// Mitsubishi GX Works2 project: BKVinaTest   PLC: FX3U/FX3UC

// global labels: Global1
VAR_GLOBAL
  ALARM AT Y012 : BOOL;
  OPERATION AT Y013 : BOOL;
  RelayXLKC1 AT Y014 : BOOL;
  RelayXLC2 AT Y015 : BOOL;
  RelayXLD3_1 AT Y016 : BOOL;
  RelayXLD3_2 AT Y017 : BOOL;
  RelayXLX4_1 AT Y020 : BOOL;
  RelayXLX4_2 AT Y021 : BOOL;
  RelayXLX5_1 AT Y022 : BOOL;
  RelayXLX5_2 AT Y023 : BOOL;
  RelayXLD6_1 AT Y024 : BOOL;
  RelayLubOil AT Y025 : BOOL;
  RelayXLTT AT Y026 : BOOL;
  RelayXLTP AT Y027 : BOOL;
  RelayXLDT AT Y030 : BOOL;
  RelayXLDP AT Y031 : BOOL;
  RelayXLKDT AT Y032 : BOOL;
  RelayXLKDP AT Y033 : BOOL;
  RelayTT AT Y034 : BOOL;
  RelayMR_1 AT Y035 : BOOL;
  RelayMR_2 AT Y036 : BOOL;
  RelayMXC_1 AT Y037 : BOOL;
  RelayMXC_2 AT Y040 : BOOL;
  RelayMQ_1 AT M10 : BOOL;
  RelayMQ_2 : BOOL;
  RelayMXDT_1 AT Y041 : BOOL;
  RelayMXDT_2 AT Y042 : BOOL;
  RelayMXDP_1 AT Y043 : BOOL;
  RelayMXDP_2 AT Y044 : BOOL;
  RelayOilP AT Y045 : BOOL;
  RelayOilV1 AT Y046 : BOOL;
  RelayOilV2 AT Y047 : BOOL;
  CommandMXC_F AT M260 : BOOL;
  CommandMXC_Z AT M261 : BOOL;
  CommandMQ_F AT M262 : BOOL;
  CommandMQ_Z AT M263 : BOOL;
  CommandMXDT_F AT M264 : BOOL;
  CommandMXDT_Z AT M265 : BOOL;
  CommandMXDP_F AT M267 : BOOL;
  CommandMXDP_Z AT M268 : BOOL;
  CommandMR_L AT M269 : BOOL;
  CommandMR_R AT M270 : BOOL;
  CommandXLXC_I AT M271 : BOOL;
  CommandXLXC_O AT M272 : BOOL;
  CommandPHA_1 AT M273 : BOOL;
  CommandPHA_2 AT M274 : BOOL;
  MR_L AT X010 : BOOL;
  MR_R AT X011 : BOOL;
  CB3 AT X012 : BOOL;
  EMERG AT X013 : BOOL;
  MainRST AT X014 : BOOL;
  START AT X015 : BOOL;
  Jog_Left AT X016 : BOOL;
  Jog_Right AT X017 : BOOL;
  PushOilPump AT X020 : BOOL;
  XLKC1_I AT X021 : BOOL;
  XLKC1_O AT X022 : BOOL;
  XLC2_I AT X023 : BOOL;
  XLC2_O AT X024 : BOOL;
  XLD3_I AT X025 : BOOL;
  XLD3_O AT X026 : BOOL;
  XLX4_I AT X027 : BOOL;
  XLX4_O AT X030 : BOOL;
  XLX5_I AT X031 : BOOL;
  XLX5_O AT X032 : BOOL;
  XLD6_I AT X033 : BOOL;
  XLD6_O AT X034 : BOOL;
  XLTT_I AT X035 : BOOL;
  XLTP_I AT X036 : BOOL;
  XLKDT_I AT X037 : BOOL;
  XLKDP_I AT X040 : BOOL;
  XLDT_I AT X041 : BOOL;
  XLDT_O AT X042 : BOOL;
  XLDP_I AT X043 : BOOL;
  XLDP_O AT X044 : BOOL;
  OLPump AT X045 : BOOL;
  MR_L1 AT X046 : BOOL;
  MR_R1 AT X047 : BOOL;
  MXC_ZX AT X004 : BOOL;
  MQ_ZX AT X005 : BOOL;
  MXDT_ZX AT X002 : BOOL;
  MXDP_ZX AT X003 : BOOL;
  Round_MXC AT D200 : REAL;
  Round_MQL AT D202 : REAL;
  Round_MQR AT D204 : REAL;
  Round_MXDT AT D206 : REAL;
  Round_MXDP AT D208 : REAL;
  CommandBTX AT M275 : BOOL;
  CommandXLTT AT M276 : BOOL;
  CommandXLTP AT M277 : BOOL;
  CommandXLDT AT M278 : BOOL;
  CommandXLDP AT M279 : BOOL;
  CommandXLKC1 AT M280 : BOOL;
  CommandXLC2 AT M281 : BOOL;
  MXC_Z AT M282 : BOOL;
  MQ_Z AT M283 : BOOL;
  MXDT_Z AT M284 : BOOL;
  MXDP_Z AT M285 : BOOL;
  MXC_FWD AT M286 : BOOL;
  MQ_FWD AT M287 : BOOL;
  MXDT_FWD AT M288 : BOOL;
  MXDP_FWD AT M289 : BOOL;
  ModeAuto : BOOL;
  StopEmerg : BOOL;
  activeCK : BOOL;
  pushManXLKC1 AT M200 : BOOL;
  pushManXLC2 AT M201 : BOOL;
  pushManXLD3_I AT M202 : BOOL;
  pushManXLD3_O AT M203 : BOOL;
  pushManXLX4_I AT M204 : BOOL;
  pushManXLX4_O AT M205 : BOOL;
  pushManXLX5_I AT M206 : BOOL;
  pushManXLX5_O AT M207 : BOOL;
  pushManXLD6_I AT M208 : BOOL;
  pushManXLD6_O AT M209 : BOOL;
  pushManXLTT AT M210 : BOOL;
  pushManXLTP AT M211 : BOOL;
  pushManXLKDT AT M212 : BOOL;
  pushManXLKDP AT M213 : BOOL;
  pushManXLDT AT M214 : BOOL;
  pushManXLDP AT M215 : BOOL;
  pushManTT AT M216 : BOOL;
  pushManMXC_F AT M217 : BOOL;
  pushManMXC_Z AT M218 : BOOL;
  pushManMQ_F AT M219 : BOOL;
  pushManMQ_Z AT M220 : BOOL;
  pushManMXDT_F AT M221 : BOOL;
  pushManMXDT_Z AT M222 : BOOL;
  pushManMXDP_F AT M223 : BOOL;
  pushManMXDP_Z AT M224 : BOOL;
  PushOilV1 AT M225 : BOOL;
  PushOilV2 AT M226 : BOOL;
  pushB8 AT M227 : BOOL;
  pushB9 AT M228 : BOOL;
  pushB10 AT M229 : BOOL;
  pushCa1 AT M230 : BOOL;
  pushCa2 AT M231 : BOOL;
  pushCa3 AT M232 : BOOL;
  rstTotalB AT M233 : BOOL;
  rstCounterCK AT M234 : BOOL;
  rstAmountCK AT M235 : BOOL;
  restory AT M236 : BOOL;
  Round_MR AT D210 : REAL;
  Speed_MXC AT D212 : REAL;
  Speed_MQ AT D214 : REAL;
  Speed_MXDT AT D216 : REAL;
  Speed_MXDP AT D218 : REAL;
  Speed_MR AT D220 : REAL;
  Speed_MXCZ AT D222 : REAL;
  Speed_MQZ AT D224 : REAL;
  Speed_MXDTZ AT D226 : REAL;
  Speed_MXDPZ AT D228 : REAL;
  Speed_MRZ AT D230 : REAL;
  Real_MXC : REAL;
  Real_MQ : REAL;
  Real_MXDT : REAL;
  Real_MXDP : REAL;
  Real_MR : REAL;
  Freq_MXC : REAL;
  Freq_MQ : REAL;
  Freq_MXDT : REAL;
  Freq_MXDP : REAL;
  Freq_MR : REAL;
  TimeMR_DSL AT D240 : DWORD;
  TimeMR_R AT D242 : DWORD;
  TimeMR_E AT D244 : DWORD;
  TimeERROR AT D246 : DWORD;
  MXCF1 AT Y000 : BOOL;
  MXCE1 AT Y001 : BOOL;
  MXCD1 AT Y002 : BOOL;
  MR_DSLOW AT Y011 : BOOL;
  ca1_B8 AT D250 : DWORD;
  ca2_B8 AT D252 : DWORD;
  ca3_B8 AT D254 : DWORD;
  ca1_B9 AT D256 : DWORD;
  ca2_B9 AT D258 : DWORD;
  ca3_B9 AT D260 : DWORD;
  ca1_B10 AT D262 : DWORD;
  ca2_B10 AT D264 : DWORD;
  ca3_B10 AT D266 : DWORD;
  total_B8 AT D268 : DWORD;
  total_B9 AT D270 : DWORD;
  total_B10 AT D272 : DWORD;
  NumberCK AT D280 : DWORD;
  CounterCK AT D282 : DWORD;
  AmountCK AT D284 : DWORD;
  TotalCK AT D286 : DWORD;
  PushLubOil AT M237 : BOOL;
  Pape1 AT M240 : BOOL;
  Pape2 AT M241 : BOOL;
  Pape3 AT M242 : BOOL;
  PushPause AT M238 : BOOL;
  Pape0 AT M239 : BOOL;
  IndicateMXC AT D232 : REAL;
  IndicateMQ AT D234 : REAL;
  IndicateMXDT AT D236 : REAL;
  IndicateMXDP AT D238 : REAL;
END_VAR

// task Task_01 (event TRUE, interval 0, priority 31): PowerControl, StepControl
// task InterruptMXC (event I010, interval 0, priority 31): EncoderX001
// task InterruptMXDT (event I020, interval 0, priority 31): EncoderX006
// task InterruptMXDP (event I030, interval 0, priority 31): EncoderX007
// task InterruptMQ_Z (event I501, interval 0, priority 31): PickupX005
// task InterruptMXC_Z (event I400, interval 0, priority 31): PickupX004
// task InterruptMXDT_Z (event I200, interval 0, priority 31): PickupX002
// task InterruptMXDP_Z (event I300, interval 0, priority 31): PickupX003

PROGRAM PowerControl
VAR
  ButtonOilP : BOOL;
  ButtonOilV1 : BOOL;
  ButtonOilV2 : BOOL;
  MR : MotorRev;
  MQ : MotorRev;
  MXC : MotorRev;
  MXDT : MotorRev;
  MXDP : MotorRev;
  XLKC1 : MotorOne;
  XLC2 : MotorOne;
  XLD3 : MotorRev;
  XLX4 : MotorRev;
  XLX5 : MotorRev;
  XLD6 : MotorOne;
  XLTT : MotorOne;
  XLTP : MotorOne;
  XLKDT : MotorOne;
  XLKDP : MotorOne;
  XLDT : MotorOne;
  XLDP : MotorOne;
  OILPUMP : MotorOne;
  VALVE1 : MotorOne;
  VALVE2 : MotorOne;
  Servo_MXC : Servo;
  TimerMR_DSL : TON;
  TimerMRDSL_Q : BOOL;
  ManualMXC_F : BOOL;
  ManualMXC_Z : BOOL;
  ManualMQ_F : BOOL;
  ManualMQ_Z : BOOL;
  ManualMXDT_F : BOOL;
  ManualMXDT_Z : BOOL;
  ManualMXDP_F : BOOL;
  ManualMXDP_Z : BOOL;
  Dint_C251 : DINT;
  Dint_C234 : DINT;
  Dint_C244 : DINT;
  Dint_C245 : DINT;
END_VAR
EI( TRUE );
(* MR: Chạy khi cụm xoắn đầu chạy *)
MR(SetAutoMan := ModeAuto, PushManF := Jog_Left , PushManR := Jog_Right ,
		LimitInputF := NOT MR_L OR NOT TimerMRDSL_Q, LimitInputR := NOT MR_R OR NOT TimerMRDSL_Q,
		SetAutoRunF := CommandMR_L, SetAutoRunR := CommandMR_R ,
		OutputF := RelayMR_1, OutputR:= RelayMR_2);

RelayTT := (RelayMR_1 AND NOT MR_L) OR (RelayMR_2 AND NOT MR_R);
TimerMR_DSL(IN := (NOT MR_L AND RelayMR_1) OR (NOT MR_R AND RelayMR_2), 
								PT := DWORD_TO_TIME(TimeMR_DSL), Q := TimerMRDSL_Q );

SET(LDP(TRUE, (MR_L1 AND RelayMR_1) OR (MR_R1 AND RelayMR_2)), MR_DSLOW);
RST(LDP(TRUE, RelayMR_1 OR RelayMR_2), MR_DSLOW);

(* MXQ: *)
(* Initialize FX2N-1HC => MQ control *)
TO( M8002, K0, K0 , K0, K1 );
DTO( M8002, K2147483647, K0 , K2, K1 );
DTO( M8002 , REAL_TO_DINT( Real_MQ ) , K0, K12 , K1);

M11 := ModeAuto;
M13 := ModeAuto;
M10 := CommandMQ_F OR pushManMQ_F;
M14 := NOT M10;
SET( LDP(TRUE, M10), M22); (*YS output set *)
RST( LDF(TRUE, M34), M8055);
RST( LDF(TRUE, M34), CommandMQ_F);

TO( TRUE, K4M10, K0 , K4, K1 );
DFROM( TRUE, K0 , K20 , K1, C234 );
FROM( ModeAuto, K0 , K27 , K1 , K3M30 );
DTO( LDF(TRUE, M10) , K0 , K0, K20 , K1); (* software reset counter *)

(*Manual*)	

RST( LDF(TRUE , NOT ModeAuto AND pushManMQ_F), M20); (*YS output reset*)
	
(* MXC:  CommandXLXC_I  and CommandXLXC_O *)	
SET( LDP(TRUE, XLD3_O AND XLX4_O), CommandMXC_F);
MXC(SetAutoMan:= ModeAuto, PushManF := pushManMXC_F, 
			LimitInputF := MXC_FWD, LimitInputR := MXC_Z,
			SetAutoRunF := CommandMXC_F, SetAutoRunR := CommandMXC_Z,
			OutputF := RelayMXC_1, OutputR := RelayMXC_2);

RST( LDP(TRUE, CommandXLXC_O), CommandXLXC_I);
RST( LDF(TRUE, CommandMXC_Z), CommandXLXC_O);
SET( LDF(TRUE, CommandMXC_Z), CommandXLXC_I);
XLD3(SetAutoMan := ModeAuto,
			PushManF := pushManXLD3_O, PushManR := pushManXLD3_I,
			LimitInputF := TRUE, LimitInputR := TRUE,
			SetAutoRunF := CommandXLXC_O, SetAutoRunR := CommandXLXC_I,
			OutputF := RelayXLD3_1, OutputR := RelayXLD3_2);			
			
XLX4(SetAutoMan := ModeAuto,
			PushManF := pushManXLX4_O, PushManR := pushManXLX4_I,
			LimitInputF := TRUE , LimitInputR := TRUE,
			SetAutoRunF := CommandXLXC_O, SetAutoRunR := CommandXLXC_I,
			OutputF := RelayXLX4_1, OutputR := RelayXLX4_2);				
	
(* MXDT:  CommandXLDT => dừng khi encoder đủ vòng *)	
SET( LDP(TRUE, XLDT_O), CommandMXDT_F);
SET( LDP(TRUE, XLDT_I), CommandMXDT_Z);
MXDT(SetAutoMan := ModeAuto, PushManF := pushManMXDT_F, 
			LimitInputF := MXDT_FWD, LimitInputR := MXDT_Z,
			SetAutoRunF :=  CommandMXDT_F, SetAutoRunR := CommandMXDT_Z ,
			OutputF := RelayMXDT_1, OutputR := RelayMXDT_2);

RST( LDF(TRUE, MXDT_FWD), CommandXLDT);
XLKDT(SetAutoMan := ModeAuto, 
			PushMan := pushManXLKDT, LimitInput :=  TRUE,
			SetAutoRun := CommandXLDT, Output := RelayXLKDT);

XLDT(SetAutoMan := ModeAuto, 
			PushMan := pushManXLDT, LimitInput :=TRUE,
			SetAutoRun := CommandXLDT, Output := RelayXLDT);	

(* MXDP:  CommandXLDP => dừng khi encoder đủ vòng *)	
SET( LDP(TRUE, XLDP_O), CommandMXDP_F);
SET( LDP(TRUE, XLDP_I), CommandMXDP_Z);
MXDP(SetAutoMan := ModeAuto, PushManF := pushManMXDP_F, 
			LimitInputF := MXDP_FWD, LimitInputR := MXDP_Z,
			SetAutoRunF := CommandMXDP_F, SetAutoRunR := CommandMXDP_Z ,
			OutputF := RelayMXDP_1, OutputR := RelayMXDP_2);

RST( LDF(TRUE, MXDP_FWD), CommandXLDP);
XLKDP(SetAutoMan := ModeAuto, 
			PushMan := pushManXLKDP, LimitInput := TRUE,
			SetAutoRun := CommandXLDP, Output := RelayXLKDP);
			
XLDP(SetAutoMan := ModeAuto,
			PushMan := pushManXLDP, LimitInput := TRUE,
			SetAutoRun := CommandXLDP, Output := RelayXLDP);

(* PHA:  CommandPHA_1  and CommandPHA_2 *)	
SET(LDP(TRUE, MR_R AND CommandBTX), CommandPHA_1);
SET(LDP(TRUE, MR_L AND CommandBTX), CommandPHA_2);	
XLX5(SetAutoMan := ModeAuto,
			PushManF := pushManXLX5_O, PushManR := pushManXLX5_I,
			LimitInputF := TRUE , LimitInputR := TRUE,
			SetAutoRunF := CommandPHA_1, SetAutoRunR := CommandPHA_2,
			OutputF := RelayXLX5_1, OutputR := RelayXLX5_2);				
			
XLD6(SetAutoMan := ModeAuto,
			PushMan := pushManXLD6_O, LimitInput := TRUE ,
			SetAutoRun := CommandPHA_1, Output := RelayXLD6_1);				

(* BTX:  CommandBTX  *)
RST(LDP(TRUE, CommandBTX), CommandXLKC1);
SET(LDP(TRUE, CommandBTX), CommandXLC2);
SET(LDP(TRUE,XLC2_O), CommandXLKC1);
RST(LDP(TRUE,XLKC1_O), CommandBTX);
XLKC1(SetAutoMan := ModeAuto,
			PushMan := pushManXLKC1, LimitInput := TRUE,
			SetAutoRun := CommandXLKC1, Output := RelayXLKC1);

XLC2(SetAutoMan := ModeAuto,
			PushMan := pushManXLC2, LimitInput := NOT XLKC1_I OR NOT ModeAuto,
			SetAutoRun := CommandXLC2, Output := RelayXLC2);
			
(* TLT: CommandXLTT => chạy theo cylinder  xoắn đầu *)
SET( LDP(TRUE, XLDT_O), CommandXLTT);
XLTT(SetAutoMan := ModeAuto,
			PushMan := pushManXLTT, LimitInput := MXDT_FWD OR NOT ModeAuto,
			SetAutoRun := CommandXLTT, Output := RelayXLTT);
			
(* TLP: CommandXLTP => chạy theo cylinder  xoắn đầu *)
SET( LDP(TRUE, XLDP_O), CommandXLTP);
XLTP(SetAutoMan := ModeAuto, 
			PushMan := pushManXLTP, LimitInput := MXDP_FWD OR NOT ModeAuto,
			SetAutoRun := CommandXLTP, Output := RelayXLTP);

(* Hydrolic control *)
ButtonOilP := LDP(TRUE, PushOilPump) XOR ButtonOilP;
OILPUMP(PushMan := ButtonOilP, LimitInput := NOT OLPump, Output := RelayOilP );

RelayOilV1 := RelayMQ_1 OR RelayMXDP_1 OR RelayMXDP_2 OR RelayMXDT_1 OR RelayMXDT_2 OR RelayXLX5_1 OR RelayXLX5_2;
RelayOilV2 := RelayMXC_1 OR RelayMXC_2 OR RelayXLD3_1 OR RelayXLD3_2 OR RelayXLX4_1 OR RelayXLX4_2;
RelayLubOil := LDP(TRUE, PushLubOil) XOR RelayLubOil;

IF ModeAuto THEN
	(* Forward at Zero *)
	SET( CommandMXC_F AND X004, MXC_FWD);
	SET( CommandMXDT_F AND X002, MXDT_FWD);
	SET( CommandMXDP_F AND X003, MXDP_FWD);
	
	(* Set Home *)
	SET( LDF(TRUE, RelayMXC_1), CommandMXC_Z);
	SET( LDF(TRUE, XLDT_I), CommandMXDT_Z);
	SET( LDF(TRUE, XLDP_I), CommandMXDP_Z);
	
	SET( LDF(TRUE, RelayMXC_1), MXC_Z);
	SET( LDF(TRUE, RelayMXDT_1), MXDT_Z);
	SET( LDF(TRUE, RelayMXDP_1), MXDP_Z);
	
	(* Set Interrupt *)
	RST( LDP(TRUE, RelayMXC_2), M8054);
	RST( LDP(TRUE, RelayMXDT_2), M8052);
	RST( LDP(TRUE, RelayMXDP_2), M8053);
ELSE	
	SET( LDP(TRUE, pushManMXC_F), MXC_FWD);
	SET( LDP(TRUE, pushManMXDT_F), MXDT_FWD);
	SET( LDP(TRUE, pushManMXDP_F), MXDP_FWD);
END_IF;

(* initialize encoder interrupt *)
RST( LDP(TRUE, RelayMXC_1), C251);
RST( LDP(TRUE, RelayMXDT_1), C244);
RST( LDP(TRUE, RelayMXDP_1), C245);
M8390 := M8388;
M8391 := M8388;

DWORD_TO_DINT_E( TRUE , C251 , Dint_C251 );
DWORD_TO_DINT_E( TRUE , C234 , Dint_C234 );
DWORD_TO_DINT_E( TRUE , C244 , Dint_C244 );
DWORD_TO_DINT_E( TRUE , C245 , Dint_C245 );

DEDIV( TRUE , DINT_TO_REAL(Dint_C251) , 2000.0 , D232 );
DEDIV( TRUE , DINT_TO_REAL(Dint_C234) , 360.0 , D234 );
DEDIV( TRUE , DINT_TO_REAL(Dint_C244) , 360.0 , D236 );
DEDIV( TRUE , DINT_TO_REAL(Dint_C245) , 360.0 , D238 );

(* Initialize high speed counter *)
OUT_C_32( TRUE, CC251, K2147483647);
OUT_C_32( TRUE, CC244, K2147483647);
OUT_C_32( TRUE, CC245, K2147483647);

(* Initialize high speed counter *)
DHSCS_I( TRUE , REAL_TO_DINT( Real_MXC ), CN251, I010);
DHSCS_I( TRUE , REAL_TO_DINT( Real_MXDT ), CN244, I020);
DHSCS_I( TRUE , REAL_TO_DINT( Real_MXDP ), CN245, I030);
END_PROGRAM

FUNCTION_BLOCK MotorRev
VAR_INPUT
  SetAutoMan : BOOL;
END_VAR
VAR_IN_OUT
  PushManF : BOOL;
  PushManR : BOOL;
END_VAR
VAR_INPUT
  LimitInputF : BOOL;
  LimitInputR : BOOL;
END_VAR
VAR_IN_OUT
  SetAutoRunF : BOOL;
  SetAutoRunR : BOOL;
END_VAR
VAR_OUTPUT
  OutputF : BOOL;
  OutputR : BOOL;
END_VAR
VAR
  RelayBufferF : BOOL;
  RelayBufferR : BOOL;
END_VAR
(* Set mode Auto/Man *)
IF  SetAutoMan THEN
	RelayBufferF := 	NOT SetAutoRunR AND SetAutoRunF;
	RelayBufferR := NOT SetAutoRunF AND SetAutoRunR;
ELSE
	RelayBufferF := NOT PushManR AND PushManF;
	RelayBufferR := NOT PushManF AND PushManR;
END_IF;

OutputF := RelayBufferF AND LimitInputF ;
OutputR := RelayBufferR AND LimitInputR ;
(* Reset control signal *)
RST( LDF( TRUE, OutputF) , SetAutoRunF );
RST( LDF( TRUE, OutputR) , SetAutoRunR );
END_FUNCTION_BLOCK

PROGRAM StepControl
VAR
  FistScan : BOOL;
  pushA : R_TRIG;
  flash_Status0 : R_TRIG;
  flashEmerg : F_TRIG;
  Emergency : BOOL;
  AutoEnable : BOOL;
  Error : ARRAY [0..18] OF BOOL;
  status : ARRAY [0..9] OF BOOL;
  cond : ARRAY [0..9] OF BOOL;
  count : INT;
  pointer : INT;
  TimerMRR_Q : BOOL;
  TimerMRE_Q : BOOL;
  TimerERROR_Q : BOOL;
  TimerMR_L : TON_10;
  TimerRestore : TON;
  TimerMR_E : TON;
  TimerERROR : TON;
  AuxCylinder : BOOL;
  MainCylinder : BOOL;
  TimerRestore_Q : BOOL;
END_VAR
(*
Thake production line project: Mr. Cang - Mr. Nguyen Tuan Nam
Code and graphic designer: HadiMadu - Techwaves Co,.Ltd
*)
Emergency := EMERG;

ALARM :=  Emergency OR OLPump OR TimerERROR_Q OR TimerMRE_Q;
OPERATION := status[1] OR status[2] OR status[3] OR status[4] OR status[5] OR status[6];

IF ALARM THEN
	ModeAuto := FALSE;
ELSIF MainRST THEN
	ModeAuto := TRUE;
END_IF;

(* Mode Auto *)
AutoEnable := ModeAuto AND CB3 AND NOT PushPause;

Pape0 := NOT(Pape1 OR Pape2  OR Pape3);
Pape1 := status[0] OR status[1] OR status[2];
Pape2 := status[3] OR status[4];
Pape3 := status[5] OR status[6];

(* Power control *)
AuxCylinder := XLTT_I AND XLTP_I  AND XLKDT_I AND XLKDP_I; 
MainCylinder := XLD3_I AND XLX4_I  AND XLDT_I  AND XLDP_I;

cond[0] := pointer = 0 AND AutoEnable AND MR_L AND XLD6_O AND XLX5_O AND MQ_ZX AND START; 	(* S1: Điều kiện chạy MQ*)
cond[1] := pointer = 1 AND AutoEnable AND LDP(TRUE, MQ_Z) AND MainCylinder AND AuxCylinder;		(* S2: Điều kiện chạy BXT*)
cond[2] := pointer = 2 AND AutoEnable AND LDP(TRUE, XLKC1_O);  						(* S3: Điều kiện chạy MXDT, MR-L*)
cond[3] := pointer = 3 AND AutoEnable AND LDP(TRUE, MainCylinder AND AuxCylinder); 			(* S4: Điều kiện chạy BXT, PHA 2*)
cond[4] := pointer = 4 AND AutoEnable AND LDP(TRUE, XLD6_I AND XLX5_I AND XLKC1_O AND MXDT_ZX); 	(* S5: Điều kiện chạy MXDP, MR-R*)
cond[5] := pointer = 5 AND AutoEnable AND LDP(TRUE, MainCylinder AND AuxCylinder); 			(* S6: Điều kiện chạy BXT, PHA 1*)
cond[6] := pointer = 6 AND AutoEnable AND LDP(TRUE, XLD6_O AND XLX5_O AND XLKC1_O AND MXDT_ZX); 	(* S3: Điều kiện chạy MXDT, MR-L*)

	(*cycle program*)
SET(LDP(TRUE, ModeAuto), status[0]);
IF ModeAuto THEN 
	FOR count := 0 TO 6 DO
		IF (count = 0) AND cond[0] THEN
			pointer := 1;
			status[pointer] := 1;
		END_IF;
		IF (count = 1) AND cond[1] THEN
			pointer := 2;
			status[pointer] := 1;
		END_IF;
		IF (count = 2) AND cond[2] THEN
			pointer := 3;
			status[pointer] := 1;
		END_IF;
		IF (count = 3) AND cond[3] THEN
			pointer := 4;
			status[pointer] := 1;
		END_IF;
		IF (count = 4) AND cond[4] THEN
			pointer := 5;
			status[pointer] := 1;
		END_IF;
		IF (count = 5) AND cond[5] THEN
			pointer := 6;
			status[pointer] := 1;
		END_IF;
		IF (count = 6) AND cond[6] THEN
			pointer := 3;
			status[pointer] := 1;
		END_IF;
		IF (count <> pointer) THEN
			status[count] := 0;
		END_IF;				
	END_FOR;
END_IF;

SET(LDP(TRUE, status[1]), CommandMQ_F); 
SET(LDP(TRUE, status[2] OR status[4]) OR status[6], CommandBTX); 
SET(LDP(TRUE, status[6]), CommandPHA_1); 
SET(LDP(TRUE, status[4]), CommandPHA_2); 
SET(LDP(TRUE, status[3] OR status[5]) AND (CounterCK < NumberCK), CommandXLXC_O); 
SET(LDP(TRUE, status[3]), CommandXLDT); 
SET(LDP(TRUE, status[5]), CommandXLDP); 
SET( LDP(TRUE, (MR_L AND status[3]) OR (MR_R AND status[5])), CommandMQ_F);
SET(LDP(TRUE, NOT MR_L AND status[3]), CommandMR_L);
SET(LDP(TRUE, NOT MR_R AND status[5]), CommandMR_R);

TimerMR_E(IN := RelayMR_1 OR RelayMR_2,
						PT := DWORD_TO_TIME( TimeMR_E) *1000, Q := TimerMRE_Q);						

(*Control status 0*)
IF Status[0] THEN
	SET(NOT MXC_ZX, CommandMXC_Z);
	SET(NOT MQ_ZX, CommandMQ_Z);
	SET(NOT MXDT_ZX, CommandMXDT_Z);
	SET(NOT MXDP_ZX, CommandMXDP_Z);
	SET(NOT MR_L, CommandMR_L);
	SET(NOT (XLX5_O AND XLD6_O), CommandPHA_1); 
	SET( NOT (XLD3_I AND XLX4_I) AND MXC_ZX, CommandXLXC_I); 
	RST(NOT XLDT_I, CommandXLDT); 
	RST(NOT XLDP_I, CommandXLDP); 
	RST(NOT XLC2_I, CommandXLC2);
	RST(NOT XLKC1_I, CommandXLKC1);
	RST(NOT XLTT_I, CommandXLTT); 
	RST(NOT XLDT_I, CommandXLTP); 
	RST(NOT XLKDT_I, CommandXLDT); 
	RST(NOT XLKDP_I, CommandXLDP); 
END_IF;

Error[0] := Error[1] OR Error[2] OR Error[3] OR Error[4] OR Error[5] OR Error[6] OR Error[7] OR Error[8] OR Error[9]
 					OR Error[10] OR Error[11] OR Error[12] OR Error[13] OR Error[14] OR Error[15] OR Error[16];
 					
TimerERROR(IN := Error[0], PT := DWORD_TO_TIME( TimeERROR)*1000, Q := TimerERROR_Q);

Error[1] := (RelayXLKC1 AND XLKC1_I) OR (RelayXLKC1 AND NOT XLKC1_O);
Error[2] := (RelayXLC2 AND XLC2_I) OR (RelayXLC2 AND NOT XLC2_O );
Error[3] := (RelayXLD3_1 AND XLD3_I) OR (RelayXLD3_2 AND XLD3_O);
Error[4] := (RelayXLX4_1 AND XLX4_I) OR (RelayXLX4_2 AND XLX4_O);
Error[5] := (RelayXLX5_1 AND XLX5_I) OR (RelayXLX5_2 AND XLX5_O);
Error[6] := (RelayXLD6_1 AND XLD6_I) OR (NOT RelayXLD6_1 AND XLD6_O);
Error[7] := (RelayXLDT AND XLDT_I) OR (RelayXLDT AND NOT XLDT_O);
Error[8] := (RelayXLDP AND XLDP_I) OR (RelayXLDP AND NOT XLDP_O);
Error[9] := (RelayXLKDT AND XLKDT_I);
Error[10] := (RelayXLKDP AND XLKDP_I);
Error[11] := (RelayXLTT AND XLTT_I);
Error[12] := (RelayXLTP AND XLTP_I);
Error[13] := NOT CommandMQ_Z AND MQ_ZX;
Error[14] := NOT CommandMXC_Z AND MXC_ZX;
Error[15] := NOT CommandMXDT_Z AND MXDT_ZX;
Error[16] := NOT CommandMXDP_Z AND MXDP_ZX;

TimerRestore(IN := restory, PT:= T#10s, Q := TimerRestore_Q);
IF TimerRestore_Q THEN
	Round_MQL := 1.5;
	Round_MQR := 1.5;
	Round_MXC := 2.0;
	Round_MXDT := 2.7;
	Round_MXDP := 2.7;
	NumberCK := 44;
	TimeERROR := 10;
	TimeMR_DSL := 200;
	TimeMR_E := 10;
END_IF;

(* Khai bao vong quay cho MXC *)
DEMUL( TRUE, E2000.0, Round_MXC , Real_MXC);
(* Khai báo vòng quay cho MQ bên trái *)
DEMUL( MR_L, E360.0, Round_MQL , Real_MQ);
(* Khai báo vòng quay cho MQ bên phải *)
DEMUL( MR_R, E360.0, Round_MQR , Real_MQ);
(* Khai báo vòng quay cho MXDT *)
DEMUL( TRUE, E360.0, Round_MXDT , Real_MXDT);
(* Khai báo vòng quay cho MXDP *)
DEMUL( TRUE, E360.0, Round_MXDP , Real_MXDP);

(* Khai bao thống kê sản lượng *)
DINCP( status[6] AND XLKC1_O, CounterCK);

DINCP( pushB8 AND pushCa1 AND (CounterCK >= NumberCK), ca1_B8 );
DINCP( pushB9 AND pushCa1 AND (CounterCK >= NumberCK), ca1_B9 );
DINCP( pushB10 AND pushCa1 AND (CounterCK >= NumberCK) , ca1_B10 );
DINCP( pushB8 AND pushCa2 AND (CounterCK >= NumberCK) , ca2_B8 );
DINCP( pushB9 AND pushCa2 AND (CounterCK >= NumberCK) , ca2_B9 );
DINCP( pushB10 AND pushCa2 AND (CounterCK >= NumberCK) , ca2_B10 );
DINCP( pushB8 AND pushCa3 AND (CounterCK >= NumberCK) , ca3_B8 );
DINCP( pushB9 AND pushCa3 AND (CounterCK >= NumberCK) , ca3_B9 );
DINCP( pushB10 AND pushCa3 AND (CounterCK >= NumberCK) , ca3_B10 );
DINCP( pushB8 AND (CounterCK >= NumberCK) , total_B8 );
DINCP( pushB9 AND (CounterCK >= NumberCK) , total_B9 );
DINCP( pushB10 AND (CounterCK >= NumberCK) , total_B10 );

DINCP( CounterCK >= NumberCK , AmountCK);
RST(status[1] OR rstCounterCK OR (CounterCK >= NumberCK), CounterCK);
RST(rstAmountCK, AmountCK);

IF rstTotalB THEN
	ca1_B8 := 0;
	ca1_B9 := 0;
	ca1_B10 := 0;
	ca2_B8 := 0;
	ca2_B9 := 0;
	ca2_B10 := 0;
	ca3_B8 := 0;
	ca3_B9 := 0;
	ca3_B10 := 0;
	total_B8 := 0;
	total_B9 := 0;
	total_B10 := 0;
END_IF;
END_PROGRAM

FUNCTION_BLOCK MotorOne
VAR_INPUT
  SetAutoMan : BOOL;
  PushMan : BOOL;
  LimitInput : BOOL;
END_VAR
VAR_IN_OUT
  SetAutoRun : BOOL;
END_VAR
VAR_OUTPUT
  Output : BOOL;
END_VAR
VAR
  RelayBuffer : BOOL;
END_VAR
(* Set mode Auto / Mannual *)
IF  SetAutoMan THEN
	RelayBuffer := SetAutoRun;
ELSE 
	RelayBuffer := PushMan;
END_IF;

Output := RelayBuffer AND LimitInput ;
(* Reset control signal *)
RST( LDF( TRUE, Output ) , SetAutoRun );
END_FUNCTION_BLOCK

PROGRAM EncoderX001
RST( TRUE , MXC_FWD );
RST( TRUE , M8174 );
END_PROGRAM

PROGRAM EncoderX006
RST( TRUE , MXDT_FWD );
RST( TRUE , M8176 );
END_PROGRAM

PROGRAM EncoderX007
RST( TRUE , MXDP_FWD );
RST( TRUE , M8177 );
END_PROGRAM

PROGRAM PickupX005
SET(TRUE, M19); (*YH output reset*)
SET( TRUE, M8055);
END_PROGRAM

PROGRAM PickupX004
RST(TRUE, MXC_Z);
SET( TRUE, M8054);
END_PROGRAM

PROGRAM PickupX002
RST(TRUE, MXDT_Z);
SET( TRUE, M8052);
END_PROGRAM

PROGRAM PickupX003
RST(TRUE, MXDP_Z);
SET( TRUE, M8053);
END_PROGRAM

FUNCTION_BLOCK Servo
VAR_INPUT
  SetAutoMan : BOOL;
END_VAR
VAR_IN_OUT
  PushManF : BOOL;
  PushManR : BOOL;
END_VAR
VAR_INPUT
  Speed : DWORD;
  Range : DWORD;
END_VAR
VAR_IN_OUT
  SetAutoRunF : BOOL;
  SetAutoRunR : BOOL;
END_VAR
VAR_OUTPUT
  OutputPLS : BOOL;
  OutputDIR : BOOL;
END_VAR
VAR
  RelayPLS : BOOL;
  RelayDIR : BOOL;
END_VAR
VAR_INPUT
  LimitInputF : BOOL;
  LimitInputR : BOOL;
END_VAR
(* Set mode Auto/Man *)
IF  SetAutoMan THEN
	RelayDIR := SetAutoRunR;
	RelayPLS := SetAutoRunF XOR SetAutoRunR;
ELSE
	RelayDIR := PushManR;
	RelayPLS := PushManF XOR PushManR;
END_IF;

OutputDIR := RelayDIR ;

DPLSY( RelayPLS , Speed, Range , OutputPLS );

(* Reset control signal *)
RST( LDF( TRUE, LimitInputF ) , SetAutoRunF );
RST( LDF( TRUE, LimitInputR ) , SetAutoRunR );
END_FUNCTION_BLOCK
